// TIA Portal V20 export
FUNCTION_BLOCK "Simulation"   // FB5, LAD
// stored: MemoryReserve 100, Namespace Unit1.Em7, SetENOAutomatically false
   VAR
      Simulation_addon_Instance { S7_SetPoint := 'True'} : "Simulation_addon";
      statPulse : Bool;
   END_VAR
BEGIN

REGION Network 1: cmNgBoxLockCylinderUpDown
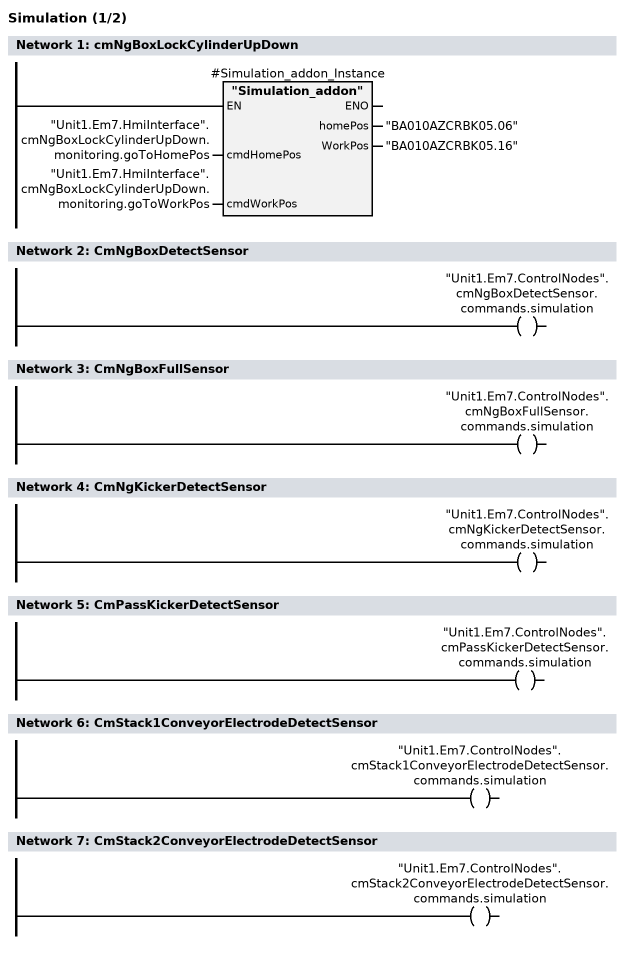
   RUNG wire#powerrail
      #Simulation_addon_Instance(cmdHomePos := "Unit1.Em7.HmiInterface".cmNgBoxLockCylinderUpDown.monitoring.goToHomePos, cmdWorkPos := "Unit1.Em7.HmiInterface".cmNgBoxLockCylinderUpDown.monitoring.goToWorkPos, homePos => "BA010AZCRBK05.06", WorkPos => "BA010AZCRBK05.16")
   END_RUNG
   // the same network as SCL:
   #Simulation_addon_Instance(cmdHomePos := "Unit1.Em7.HmiInterface".cmNgBoxLockCylinderUpDown.monitoring.goToHomePos,   // "Simulation_addon"
                           cmdWorkPos := "Unit1.Em7.HmiInterface".cmNgBoxLockCylinderUpDown.monitoring.goToWorkPos,
                           homePos => "BA010AZCRBK05.06",
                           WorkPos => "BA010AZCRBK05.16");
END_REGION

REGION Network 2: CmNgBoxDetectSensor
   RUNG wire#powerrail
      Coil( "Unit1.Em7.ControlNodes".cmNgBoxDetectSensor.commands.simulation )
   END_RUNG
   // the same network as SCL:
   "Unit1.Em7.ControlNodes".cmNgBoxDetectSensor.commands.simulation := TRUE;
END_REGION

REGION Network 3: CmNgBoxFullSensor
   RUNG wire#powerrail
      Coil( "Unit1.Em7.ControlNodes".cmNgBoxFullSensor.commands.simulation )
   END_RUNG
   // the same network as SCL:
   "Unit1.Em7.ControlNodes".cmNgBoxFullSensor.commands.simulation := TRUE;
END_REGION

REGION Network 4: CmNgKickerDetectSensor
   RUNG wire#powerrail
      Coil( "Unit1.Em7.ControlNodes".cmNgKickerDetectSensor.commands.simulation )
   END_RUNG
   // the same network as SCL:
   "Unit1.Em7.ControlNodes".cmNgKickerDetectSensor.commands.simulation := TRUE;
END_REGION

REGION Network 5: CmPassKickerDetectSensor
   RUNG wire#powerrail
      Coil( "Unit1.Em7.ControlNodes".cmPassKickerDetectSensor.commands.simulation )
   END_RUNG
   // the same network as SCL:
   "Unit1.Em7.ControlNodes".cmPassKickerDetectSensor.commands.simulation := TRUE;
END_REGION

REGION Network 6: CmStack1ConveyorElectrodeDetectSensor
   RUNG wire#powerrail
      Coil( "Unit1.Em7.ControlNodes".cmStack1ConveyorElectrodeDetectSensor.commands.simulation )
   END_RUNG
   // the same network as SCL:
   "Unit1.Em7.ControlNodes".cmStack1ConveyorElectrodeDetectSensor.commands.simulation := TRUE;
END_REGION

REGION Network 7: CmStack2ConveyorElectrodeDetectSensor
   RUNG wire#powerrail
      Coil( "Unit1.Em7.ControlNodes".cmStack2ConveyorElectrodeDetectSensor.commands.simulation )
   END_RUNG
   // the same network as SCL:
   "Unit1.Em7.ControlNodes".cmStack2ConveyorElectrodeDetectSensor.commands.simulation := TRUE;
END_REGION

REGION Network 8: Stk1 Qr Reader
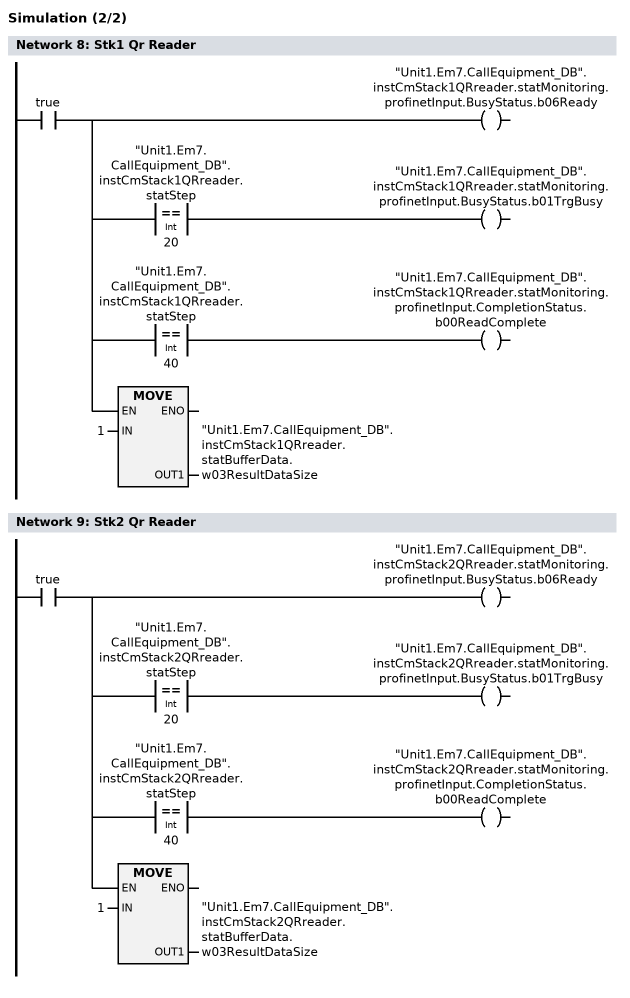
   RUNG wire#powerrail
      Contact( true )
      wire#w1
      Coil( "Unit1.Em7.CallEquipment_DB".instCmStack1QRreader.statMonitoring.profinetInput.BusyStatus.b06Ready )
   END_RUNG
   RUNG wire#w1
      { S7_Templates := "SrcType := Int" } EQ_Contact(in1 := "Unit1.Em7.CallEquipment_DB".instCmStack1QRreader.statStep, in2 := 20)
      Coil( "Unit1.Em7.CallEquipment_DB".instCmStack1QRreader.statMonitoring.profinetInput.BusyStatus.b01TrgBusy )
   END_RUNG
   RUNG wire#w1
      { S7_Templates := "SrcType := Int" } EQ_Contact(in1 := "Unit1.Em7.CallEquipment_DB".instCmStack1QRreader.statStep, in2 := 40)
      Coil( "Unit1.Em7.CallEquipment_DB".instCmStack1QRreader.statMonitoring.profinetInput.CompletionStatus.b00ReadComplete )
   END_RUNG
   RUNG wire#w1
      Move(in := 1, out1 => "Unit1.Em7.CallEquipment_DB".instCmStack1QRreader.statBufferData.w03ResultDataSize)
   END_RUNG
   // the same network as SCL:
   "Unit1.Em7.CallEquipment_DB".instCmStack1QRreader.statMonitoring.profinetInput.BusyStatus.b06Ready := true;
   "Unit1.Em7.CallEquipment_DB".instCmStack1QRreader.statMonitoring.profinetInput.BusyStatus.b01TrgBusy := true AND ("Unit1.Em7.CallEquipment_DB".instCmStack1QRreader.statStep = 20);
   "Unit1.Em7.CallEquipment_DB".instCmStack1QRreader.statMonitoring.profinetInput.CompletionStatus.b00ReadComplete := true AND ("Unit1.Em7.CallEquipment_DB".instCmStack1QRreader.statStep = 40);
   IF true THEN
       "Unit1.Em7.CallEquipment_DB".instCmStack1QRreader.statBufferData.w03ResultDataSize := 1;
   END_IF;
END_REGION

REGION Network 9: Stk2 Qr Reader
   RUNG wire#powerrail
      Contact( true )
      wire#w1
      Coil( "Unit1.Em7.CallEquipment_DB".instCmStack2QRreader.statMonitoring.profinetInput.BusyStatus.b06Ready )
   END_RUNG
   RUNG wire#w1
      { S7_Templates := "SrcType := Int" } EQ_Contact(in1 := "Unit1.Em7.CallEquipment_DB".instCmStack2QRreader.statStep, in2 := 20)
      Coil( "Unit1.Em7.CallEquipment_DB".instCmStack2QRreader.statMonitoring.profinetInput.BusyStatus.b01TrgBusy )
   END_RUNG
   RUNG wire#w1
      { S7_Templates := "SrcType := Int" } EQ_Contact(in1 := "Unit1.Em7.CallEquipment_DB".instCmStack2QRreader.statStep, in2 := 40)
      Coil( "Unit1.Em7.CallEquipment_DB".instCmStack2QRreader.statMonitoring.profinetInput.CompletionStatus.b00ReadComplete )
   END_RUNG
   RUNG wire#w1
      Move(in := 1, out1 => "Unit1.Em7.CallEquipment_DB".instCmStack2QRreader.statBufferData.w03ResultDataSize)
   END_RUNG
   // the same network as SCL:
   "Unit1.Em7.CallEquipment_DB".instCmStack2QRreader.statMonitoring.profinetInput.BusyStatus.b06Ready := true;
   "Unit1.Em7.CallEquipment_DB".instCmStack2QRreader.statMonitoring.profinetInput.BusyStatus.b01TrgBusy := true AND ("Unit1.Em7.CallEquipment_DB".instCmStack2QRreader.statStep = 20);
   "Unit1.Em7.CallEquipment_DB".instCmStack2QRreader.statMonitoring.profinetInput.CompletionStatus.b00ReadComplete := true AND ("Unit1.Em7.CallEquipment_DB".instCmStack2QRreader.statStep = 40);
   IF true THEN
       "Unit1.Em7.CallEquipment_DB".instCmStack2QRreader.statBufferData.w03ResultDataSize := 1;
   END_IF;
END_REGION
END_FUNCTION_BLOCK
